(*
Implements the procedure for safely transitioning between device states by asserting the correct beam parameters for 
the state *)
FUNCTION_BLOCK BeamClassTransitionManager
VAR_INPUT
	i_TransitionAssertionID	:	INT := 0;
	i_stTransitionAssertion : ST_BeamParams := PMPS_GVL_BeamParams.cstSafeBeam; //Assertion required during transition (always safer than anything inbetween)
	
	i_nRequestedAssertionID	:	INT := 0;
	i_stRequestedAssertion	:	ST_BeamParams := PMPS_GVL_BeamParams.cstSafeBeam; //Requested assertion, change whenever
	
	i_xMoving	:	BOOL := FALSE; //Provide rising edge when device begins moving
	i_xDoneMoving	:	BOOL := FALSE; //Provide rising edge when device is done with a move
	i_stFullBeam	:	ST_BeamParams := PMPS_GVL_BeamParams.cstFullBeam; //Beam parameters applied to transition assertion once transition is complete
END_VAR
VAR_OUTPUT
	
	q_stTransitionAssertion	:	ST_BeamParams; //Transition assertion, connect to arbiter
	q_stFinalAssertion	:	ST_BeamParams; //Final assertion, connect to arbiter
	q_xTransitionAuthorized	:	BOOL := FALSE; //Rising edge indicating the device is safe to move, use as input to move execute (which requires a rising edge)
END_VAR
VAR
	stTargetAssertion	:	ST_BeamParams; //Current target assertion
	thing	:	BOOL;
	
	xNewBP	:	BOOL;
	xTranBP	:	BOOL;
	xFinalBP	:	BOOL;
	
END_VAR

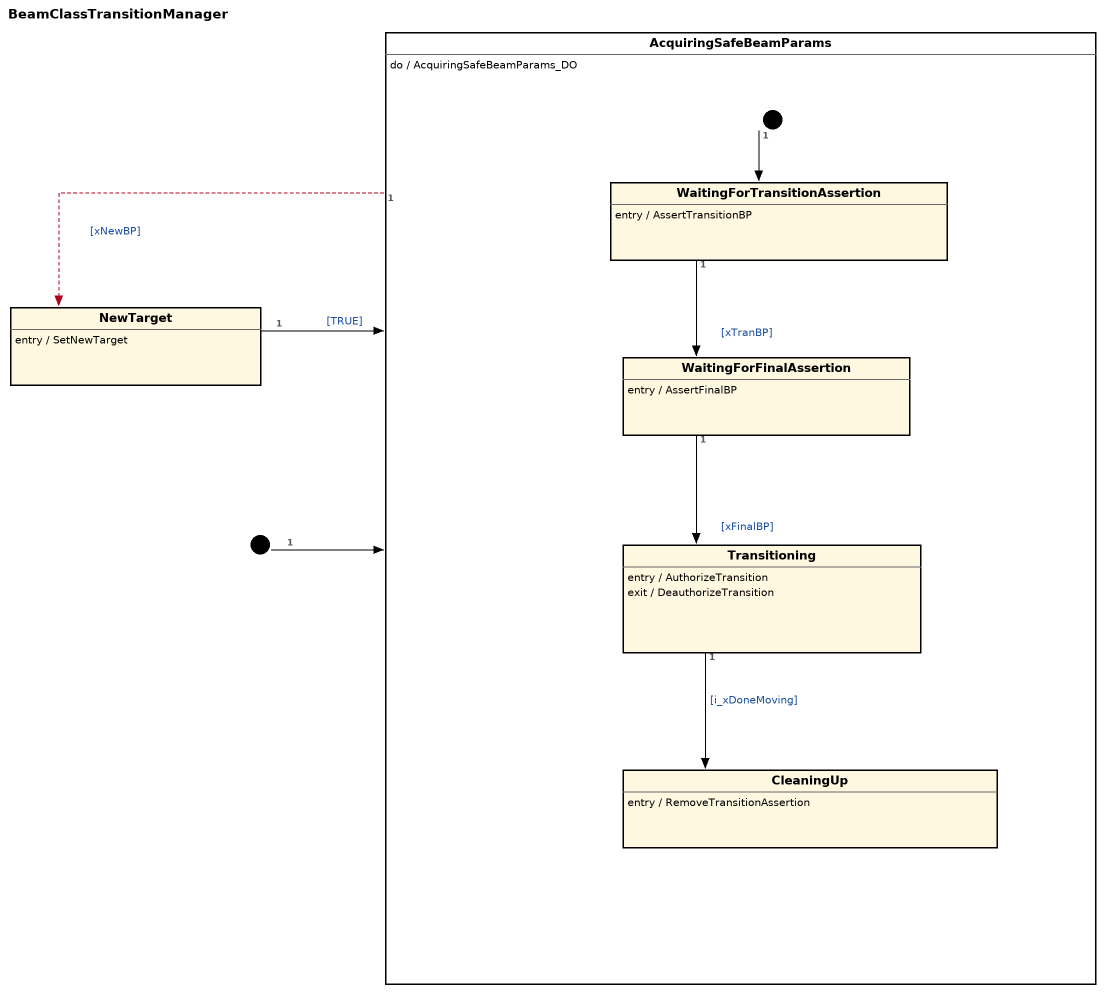
STATECHART BeamClassTransitionManager_1  // abortable
    START StartState1_copy
    COMPOSITE STATE AcquiringSafeBeamParams
        do / AcquiringSafeBeamParams_DO
        START StartState1
        STATE WaitingForTransitionAssertion
            entry / AssertTransitionBP
        STATE WaitingForFinalAssertion
            entry / AssertFinalBP
        STATE Transitioning
            entry / AuthorizeTransition
            exit / DeauthorizeTransition
        STATE CleaningUp
            entry / RemoveTransitionAssertion
        StartState1 -> WaitingForTransitionAssertion  // priority 1, on completion
        WaitingForTransitionAssertion -> WaitingForFinalAssertion [xTranBP] // priority 1
        WaitingForFinalAssertion -> Transitioning [xFinalBP] // priority 1
        Transitioning -> CleaningUp [i_xDoneMoving] // priority 1, rising edge
    END_STATE
    STATE NewTarget
        entry / SetNewTarget
    StartState1_copy -> AcquiringSafeBeamParams  // priority 1, on completion
    AcquiringSafeBeamParams -> NewTarget [xNewBP] // priority 1, exception, rising edge
    NewTarget -> AcquiringSafeBeamParams [TRUE] // priority 1
END_STATECHART

ACTION AcquiringSafeBeamParams_DO:
xNewBP := F_DifferentBeamParams(stTargetAssertion, i_stRequestedAssertion);
xTranBP	:= F_SafeBPCompare(PMPS_GVL_BeamParams.stCurrentBeamParameters, i_stTransitionAssertion);
xFinalBP := F_SafeBPCompare(PMPS_GVL_BeamParams.stCurrentBeamParameters, stTargetAssertion);
END_ACTION

ACTION AssertFinalBP:
q_stFinalAssertion := stTargetAssertion;
END_ACTION

ACTION AssertTransitionBP:
q_stTransitionAssertion := i_stTransitionAssertion;
END_ACTION

ACTION AuthorizeTransition:
q_xTransitionAuthorized := TRUE;
END_ACTION

ACTION DeauthorizeMove:

END_ACTION

ACTION DeauthorizeTransition:
q_xTransitionAuthorized := FALSE;
END_ACTION

ACTION RemoveTransitionAssertion:
q_stTransitionAssertion := PMPS_GVL_BeamParams.cstFullBeam;
END_ACTION

ACTION SetNewTarget:
stTargetAssertion := i_stRequestedAssertion;
END_ACTION

END_FUNCTION_BLOCK

(* stored: Version 1.1.0.1, ProductVersion 3.1.4022.12
   POU BeamClassTransitionManager: Id {843312b6-3630-0fa6-1e20-da1ce4aaad4c}, SpecialFunc None
   Action AcquiringSafeBeamParams_DO: Id {603c4e25-97d2-01fd-3380-8f019adaa760}
   Action AssertFinalBP: Id {3aacecc4-95cc-0b9d-1f9c-d6c9dec8e836}
   Action AssertTransitionBP: Id {09eb738b-7411-0821-2e23-c9281e93e49d}
   Action AuthorizeTransition: Id {b727a18e-e395-0e7a-074b-b778698df218}
   Action DeauthorizeMove: Id {3b9e719b-fa51-0c03-3729-27bd539c56ba}
   Action DeauthorizeTransition: Id {85553ff9-652b-0f0d-38e0-23e9eece0909}
   Action RemoveTransitionAssertion: Id {fd3da30e-395a-0698-0f23-a3f0bc8df59f}
   Action SetNewTarget: Id {cb54fd73-aaf3-0c05-2881-782da729c59b} *)
